TYPE T_Ctrl_SIf_RFW_In :
STRUCT
END_STRUCT
END_TYPE

(* stored: Version 1.1.0.1, ProductVersion 3.1.0.20
   DUT T_Ctrl_SIf_RFW_In: Id {dbc9c954-8778-46e0-8057-f6886c73fe2b} *)
